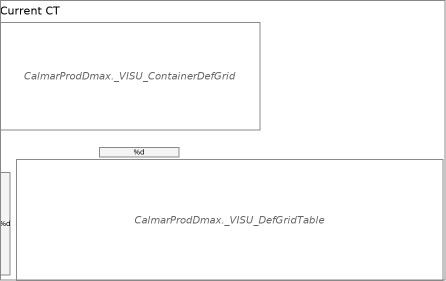
VISUALIZATION _VISU_CT_Details  // 446x281
VAR_IN_OUT
  mInst : FB_WorkerDefGrid_Deformation;
END_VAR
    Frame (0,22 260x108)
        shows CalmarProdDmax._VISU_ContainerDefGrid(m_Inst := mInst._pMultiAttachedCTs[1]^)
    Frame (16,159 427x122)
        shows CalmarProdDmax._VISU_DefGridTable(m_Inst := mInst._pMultiAttachedCTs[1]^.fBImageDeformation, m_row_start := mInst.nGridRowStart, m_col_start := mInst.nGridColStart)
    Scrollbar (99,147 80x10), "%d", text variable: mInst.nGridColStart
        p2245068023: mInst._pMultiAttachedCTs[1]^.fBImageDeformation.nMAX_ROWS_DEFGRID-2
        p1057716461: mInst.nGridColStart
    Scrollbar (0,172 10x103), "%d", text variable: mInst.nGridRowStart
        p2245068023: mInst._pMultiAttachedCTs[1]^.fBImageDeformation.nMAX_ROWS_DEFGRID
        p1057716461: mInst.nGridRowStart
    Label (-3,1 150x20), "Current CT"
END_VISUALIZATION

(* stored: Version 1.1.0.1, ProductVersion 3.1.4024.11
   Visu _VISU_CT_Details: Id {fa556a5f-0d99-4f39-a7a9-95b575bcc870} *)
